// TwinCAT 3 PLC project PLC_Pro
// ProgramVersion: 3.1.4020.4
// libraries:
//   Tc2_MC2, * (Beckhoff Automation GmbH)
//   Tc2_Standard, * (Beckhoff Automation GmbH)
//   Tc2_System, * (Beckhoff Automation GmbH)
//   Tc3_Module, * (Beckhoff Automation GmbH)
//   VisuDialogs, * (System)
// project tree:
//   / GlobalTextList.TcGTLO, PlcTask.TcTTO, 视图管理器.TcVMO (not stored)
//   POUs/ MAIN.TcPOU
//   VISUs/ HMI.TcVIS
// real-time tasks:
//   TASK Task 1: cycle T#10ms, priority 1, ADS port 350
//   TASK PlcTask: cycle T#10ms, priority 20, ADS port 351
// motion (NC):
//   TASK NC-Task 1 SAF: cycle T#2ms, priority 4, ADS port 501
//   TASK NC-Task 1 SVB: cycle T#10ms, priority 8, ADS port 511
//   AXIS Axis 1 (id 1)
//     Velo: SlowManual=0.2, FastManual=1
//     OtherSettings: AllowMotionCmdToSlave=true, PulseDistancePos=0.5, PulseDistanceNeg=0.5
//     encoder EncType=19
//       EncPara: ScaleFactorNumerator=1, ScaleFactorDenominator=10000, Inverse=true, MaxCount=#xffffffff
//     drive DrvType=16
//       DrvPara: Inverse=true, MaxCount=#xffffffff
//         TimeComp: TaskDelayCycles=1
//     controller CtrType=1
//       CtrPara: PriorControlFactor=1
//         PosDiffControl: Enable=false
//         Observer: BandWidth=20
//   AXIS Axis 2 (id 2)
//     OtherSettings: AllowMotionCmdToSlave=true
//     encoder EncType=19
//       EncPara: ScaleFactorNumerator=5, ScaleFactorDenominator=10000, MaxCount=#xffffffff
//     drive DrvType=16
//       DrvPara: MaxCount=#xffffffff
//         TimeComp: TaskDelayCycles=1
//     controller CtrType=1
//       CtrPara: PriorControlFactor=1
//         PosDiffControl: Enable=false
//         Observer: BandWidth=20
//   AXIS Axis 3 (id 3)
//     OtherSettings: AllowMotionCmdToSlave=true
//     encoder EncType=19
//       EncPara: ScaleFactorNumerator=5, ScaleFactorDenominator=10000, Inverse=true, MaxCount=#xffffffff
//     drive DrvType=16
//       DrvPara: Inverse=true, MaxCount=#xffffffff
//         TimeComp: TaskDelayCycles=1
//     controller CtrType=1
//       CtrPara: PriorControlFactor=1
//         PosDiffControl: Enable=false
//         Observer: BandWidth=20
//   AXIS Axis 4 (id 4)
//     OtherSettings: AllowMotionCmdToSlave=true
//     encoder EncType=19
//       EncPara: ScaleFactorNumerator=360, ScaleFactorDenominator=10000, MaxCount=#xffffffff
//     drive DrvType=16
//       DrvPara: MaxCount=#xffffffff
//         TimeComp: TaskDelayCycles=1
//     controller CtrType=1
//       CtrPara: PriorControlFactor=1
//         Observer: BandWidth=20
//   AXIS Axis 5 (id 5)
//     OtherSettings: AllowMotionCmdToSlave=true
//     encoder EncType=19
//       EncPara: ScaleFactorNumerator=360, ScaleFactorDenominator=10000, MaxCount=#xffffffff
//     drive DrvType=16
//       DrvPara: MaxCount=#xffffffff
//         TimeComp: TaskDelayCycles=1
//     controller CtrType=1
//       CtrPara: PriorControlFactor=1
//         PosDiffControl: Enable=false
//         Observer: BandWidth=20
// I/O:
//   DEVICE Device 2 (EtherCAT), AmsNetId 169.254.52.53.3.1
//     Drive 1 (Elmo Drive) [Gold EtherCAT GCON Drive Rev:0x00010400]
//     Drive 2 (EP3E-EC) [EP3E-EC]
//     Drive 3 (EP3E-EC) [EP3E-EC]
//     Drive 4 (EP3E-EC) [EP3E-EC]
//     Drive 5 (EP3E-EC) [EP3E-EC]
// variable links:
//   NC-Task 1 SAF/Axes/Axis 1 <-> Device 2 (EtherCAT)/Drive 1 (Elmo Drive)
//     Drive/Inputs/In/nDcOutputTime <-> InfoData/DcOutputShift
//     Drive/Inputs/In/nState1 <-> Inputs/Status word
//     Drive/Inputs/In/nState2 <-> Inputs/Status word @bit 8
//     Drive/Inputs/In/nState4 @bit 1 <-> WcState/InputToggle
//     Drive/Inputs/In/nState4 <-> WcState/WcState
//     Drive/Outputs/Out/nCtrl1 <-> Outputs/Control word
//     Drive/Outputs/Out/nCtrl2 <-> Outputs/Control word @bit 8
//     Drive/Outputs/Out/nDataOut1 <-> Outputs/Target Position
//     Enc/Inputs/In/nDataIn1 <-> Inputs/Position actual value
//     Enc/Inputs/In/nDcInputTime <-> InfoData/DcInputShift
//     Enc/Inputs/In/nState4 @bit 1 <-> WcState/InputToggle
//     Enc/Inputs/In/nState4 <-> WcState/WcState
//   NC-Task 1 SAF/Axes/Axis 2 <-> Device 2 (EtherCAT)/Drive 2 (EP3E-EC)
//     Drive/Inputs/In/nDcOutputTime <-> InfoData/DcOutputShift
//     Drive/Inputs/In/nState1 <-> 2nd Transmit PDO mapping/Statusword
//     Drive/Inputs/In/nState2 <-> 2nd Transmit PDO mapping/Statusword @bit 8
//     Drive/Inputs/In/nState4 @bit 1 <-> WcState/InputToggle
//     Drive/Inputs/In/nState4 <-> WcState/WcState
//     Drive/Outputs/Out/nCtrl1 <-> 2nd Receive PDO mapping/Controlword
//     Drive/Outputs/Out/nCtrl2 <-> 2nd Receive PDO mapping/Controlword @bit 8
//     Drive/Outputs/Out/nDataOut1 <-> 2nd Receive PDO mapping/Target Position
//     Enc/Inputs/In/nDataIn1 <-> 2nd Transmit PDO mapping/Position Actual Value
//     Enc/Inputs/In/nDcInputTime <-> InfoData/DcInputShift
//     Enc/Inputs/In/nState4 @bit 1 <-> WcState/InputToggle
//     Enc/Inputs/In/nState4 <-> WcState/WcState
//   NC-Task 1 SAF/Axes/Axis 3 <-> Device 2 (EtherCAT)/Drive 3 (EP3E-EC)
//     Drive/Inputs/In/nDcOutputTime <-> InfoData/DcOutputShift
//     Drive/Inputs/In/nState1 <-> 2nd Transmit PDO mapping/Statusword
//     Drive/Inputs/In/nState2 <-> 2nd Transmit PDO mapping/Statusword @bit 8
//     Drive/Inputs/In/nState4 @bit 1 <-> WcState/InputToggle
//     Drive/Inputs/In/nState4 <-> WcState/WcState
//     Drive/Outputs/Out/nCtrl1 <-> 2nd Receive PDO mapping/Controlword
//     Drive/Outputs/Out/nCtrl2 <-> 2nd Receive PDO mapping/Controlword @bit 8
//     Drive/Outputs/Out/nDataOut1 <-> 2nd Receive PDO mapping/Target Position
//     Enc/Inputs/In/nDataIn1 <-> 2nd Transmit PDO mapping/Position Actual Value
//     Enc/Inputs/In/nDcInputTime <-> InfoData/DcInputShift
//     Enc/Inputs/In/nState4 @bit 1 <-> WcState/InputToggle
//     Enc/Inputs/In/nState4 <-> WcState/WcState
//   NC-Task 1 SAF/Axes/Axis 4 <-> Device 2 (EtherCAT)/Drive 4 (EP3E-EC)
//     Drive/Inputs/In/nDcOutputTime <-> InfoData/DcOutputShift
//     Drive/Inputs/In/nState1 <-> 2nd Transmit PDO mapping/Statusword
//     Drive/Inputs/In/nState2 <-> 2nd Transmit PDO mapping/Statusword @bit 8
//     Drive/Inputs/In/nState4 @bit 1 <-> WcState/InputToggle
//     Drive/Inputs/In/nState4 <-> WcState/WcState
//     Drive/Outputs/Out/nCtrl1 <-> 2nd Receive PDO mapping/Controlword
//     Drive/Outputs/Out/nCtrl2 <-> 2nd Receive PDO mapping/Controlword @bit 8
//     Drive/Outputs/Out/nDataOut1 <-> 2nd Receive PDO mapping/Target Position
//     Enc/Inputs/In/nDataIn1 <-> 2nd Transmit PDO mapping/Position Actual Value
//     Enc/Inputs/In/nDcInputTime <-> InfoData/DcInputShift
//     Enc/Inputs/In/nState4 @bit 1 <-> WcState/InputToggle
//     Enc/Inputs/In/nState4 <-> WcState/WcState
//   NC-Task 1 SAF/Axes/Axis 5 <-> Device 2 (EtherCAT)/Drive 5 (EP3E-EC)
//     Drive/Inputs/In/nDcOutputTime <-> InfoData/DcOutputShift
//     Drive/Inputs/In/nState1 <-> 2nd Transmit PDO mapping/Statusword
//     Drive/Inputs/In/nState2 <-> 2nd Transmit PDO mapping/Statusword @bit 8
//     Drive/Inputs/In/nState4 @bit 1 <-> WcState/InputToggle
//     Drive/Inputs/In/nState4 <-> WcState/WcState
//     Drive/Outputs/Out/nCtrl1 <-> 2nd Receive PDO mapping/Controlword
//     Drive/Outputs/Out/nCtrl2 <-> 2nd Receive PDO mapping/Controlword @bit 8
//     Drive/Outputs/Out/nDataOut1 <-> 2nd Receive PDO mapping/Target Position
//     Enc/Inputs/In/nDataIn1 <-> 2nd Transmit PDO mapping/Position Actual Value
//     Enc/Inputs/In/nDcInputTime <-> InfoData/DcInputShift
//     Enc/Inputs/In/nState4 @bit 1 <-> WcState/InputToggle
//     Enc/Inputs/In/nState4 <-> WcState/WcState
//   PLC_Pro/PLC_Pro Instance <-> NC-Task 1 SAF/Axes/Axis 1
//     PlcTask Inputs/MAIN.motor_Line.NcToPlc <-> Outputs/ToPlc
//     PlcTask Outputs/MAIN.motor_Line.PlcToNc <-> Inputs/FromPlc
//   PLC_Pro/PLC_Pro Instance <-> NC-Task 1 SAF/Axes/Axis 2
//     PlcTask Inputs/MAIN.motor_X.NcToPlc <-> Outputs/ToPlc
//     PlcTask Outputs/MAIN.motor_X.PlcToNc <-> Inputs/FromPlc
//   PLC_Pro/PLC_Pro Instance <-> NC-Task 1 SAF/Axes/Axis 3
//     PlcTask Inputs/MAIN.motor_Y.NcToPlc <-> Outputs/ToPlc
//     PlcTask Outputs/MAIN.motor_Y.PlcToNc <-> Inputs/FromPlc
//   PLC_Pro/PLC_Pro Instance <-> NC-Task 1 SAF/Axes/Axis 4
//     PlcTask Inputs/MAIN.motor_Angle.NcToPlc <-> Outputs/ToPlc
//     PlcTask Outputs/MAIN.motor_Angle.PlcToNc <-> Inputs/FromPlc
//   PLC_Pro/PLC_Pro Instance <-> NC-Task 1 SAF/Axes/Axis 5
//     PlcTask Inputs/MAIN.motor_Master.NcToPlc <-> Outputs/ToPlc
//     PlcTask Outputs/MAIN.motor_Master.PlcToNc <-> Inputs/FromPlc
//   TcAsyncBufferReadingDrv/ReadingModule <-> TcAsyncBufferReadingDrv/WriteDetect
//     Inputs/bExecute <-> Outputs/bExecuteOut
//     Inputs/nOffset <-> Outputs/nOffset
//   TcAsyncBufferReadingDrv/WriteDetect <-> TcAsyncBufferWritingDrv/WritingModule
//     Inputs/bBusy <-> Outputs/bBusy
//     Inputs/bError <-> Outputs/bError
//     Inputs/nBytesWritten <-> Outputs/nBytesWritten

CONFIGURATION PLC_Pro
    RESOURCE PLC ON TwinCAT3
        TASK PlcTask(INTERVAL := T#10ms, PRIORITY := 20);
        PROGRAM MAIN WITH PlcTask : MAIN;
    END_RESOURCE
END_CONFIGURATION

// ---- POUs/MAIN.TcPOU
PROGRAM MAIN
VAR
	power_On_motor_All                   :BOOL :=FALSE;   (*************)
	power_On_motor_Line                  :BOOL :=FALSE; 
	power_On_motor_X                     :BOOL :=FALSE; 
    power_On_motor_Y                     :BOOL :=FALSE; 
    power_On_motor_Angle                 :BOOL :=FALSE; 
    power_On_motor_Master                :BOOL :=FALSE; 
	
	
	move_do_Line                         :BOOL :=FALSE;   (*************)
	move_do_X                            :BOOL :=FALSE;
	move_do_Y                            :BOOL :=FALSE;
    move_do_Angle                        :BOOL :=FALSE;
    move_do_Master                       :BOOL :=FALSE;
	
	set_do_Line                         :BOOL :=FALSE;    (*************)
	set_do_X                            :BOOL :=FALSE;
	set_do_Y                            :BOOL :=FALSE;
    set_do_Angle                        :BOOL :=FALSE;
    set_do_Master                       :BOOL :=FALSE;
	
	stop_do_Line                         :BOOL :=FALSE;
	stop_do_X                            :BOOL :=FALSE;
	stop_do_Y                            :BOOL :=FALSE;
    stop_do_Angle                        :BOOL :=FALSE;
    stop_do_Master                       :BOOL :=FALSE;
	
	reset_do_Line                         :BOOL :=FALSE;
	reset_do_X                            :BOOL :=FALSE;
	reset_do_Y                            :BOOL :=FALSE;
    reset_do_Angle                        :BOOL :=FALSE;
    reset_do_Master                       :BOOL :=FALSE;
	
	move_r_INC_motor_Line                 : REAL       :=0;   (****定义运动增量****)
	move_r_INC_motor_X                    : REAL       :=0;   (****关联到HMI界面****)
	move_r_INC_motor_Y                    : REAL       :=0;
	move_r_INC_motor_Angle                : REAL       :=0;
	move_r_INC_motor_Master               : REAL       :=0;
	
	(***定义轴变量***)
	motor_Line , motor_X , motor_Y , motor_Angle , motor_Master    :axis_ref;  (***定义轴变量***)
	(*****定义电源控制变量*****)
	mc_power_Line , mc_power_X , mc_power_Y , mc_power_Angle , mc_power_Master    :mc_power;   
	(****定义轴增量运动功能块*****)
	move_r_Line,  move_r_X,  move_r_Y,  move_r_Angle, move_r_Master   :mc_MoveRelative; 
	(******定义轴当前位置*****)
	position_Line, position_X, position_Y, 	position_Angle, position_Master  :mc_setposition; 
	(******定义轴停止*****) 
    stop_Line, stop_X, stop_Y, 	stop_Angle, stop_Master  :mc_stop;  
	(******定义轴复位*****)
    reset_Line, reset_X, reset_Y, reset_Angle, reset_Master  :mc_reset;  
	
END_VAR

(***********定义直线电机电源************)
mc_power_Line(
	Axis:= motor_Line, 
	Enable:= power_On_motor_All AND power_On_motor_Line, 
	Enable_Positive:= TRUE , 
	Enable_Negative:= TRUE, 
//	Override:= , 
//	BufferMode:= , 
//	Options:= , 
//	Status=> , 
//	Busy=> , 
//	Active=> , 
//	Error=> , 
//	ErrorID=> 
);
(***********定义X轴电机电源************)
	mc_power_X(
	Axis:=motor_X , 
	Enable:=power_On_motor_All AND  power_On_motor_X, 
	Enable_Positive:= TRUE, 
	Enable_Negative:= TRUE, 
	Override:= , 
	BufferMode:= , 
	Options:= , 
	Status=> , 
	Busy=> , 
	Active=> , 
	Error=> , 
	ErrorID=> );

(***********定义Y轴电机电源************)	
	mc_power_Y(
	Axis:= motor_Y, 
	Enable:= power_On_motor_All AND power_On_motor_Y, 
	Enable_Positive:= TRUE , 
	Enable_Negative:= TRUE , 
	Override:= , 
	BufferMode:= , 
	Options:= , 
	Status=> , 
	Busy=> , 
	Active=> , 
	Error=> , 
	ErrorID=> );
	
(***********定义摆角电机电源************)	
	mc_power_Angle(
	Axis:= motor_Angle, 
	Enable:=power_On_motor_All AND  power_On_motor_Angle, 
	Enable_Positive:= TRUE, 
	Enable_Negative:= TRUE, 
	Override:= , 
	BufferMode:= , 
	Options:= , 
	Status=> , 
	Busy=> , 
	Active=> , 
	Error=> , 
	ErrorID=> );
	
(***********定义主轴电机电源************)
	mc_power_Master(
	Axis:= motor_Master, 
	Enable:= power_On_motor_All AND   power_On_motor_Master, 
	Enable_Positive:= TRUE, 
	Enable_Negative:= TRUE, 
	Override:= , 
	BufferMode:= , 
	Options:= , 
	Status=> , 
	Busy=> , 
	Active=> , 
	Error=> , 
	ErrorID=> );
	
(***********定义直线电机运动************)
	move_r_Line(
	Axis:= motor_X, 
	Execute:= move_do_X, 
	Distance:= 1, 
	Velocity:=1 , 
	Acceleration:= , 
	Deceleration:= , 
	Jerk:= , 
	BufferMode:= , 
	Options:= , 
	Done=> , 
	Busy=> , 
	Active=> , 
	CommandAborted=> , 
	Error=> , 
	ErrorID=> );
	
(***********定义X轴电机运动************)
	move_r_X(
	Axis:= motor_X, 
	Execute:= move_do_X, 
	Distance:= aa, 
	Velocity:= 1, 
	Acceleration:= , 
	Deceleration:= , 
	Jerk:= , 
	BufferMode:= , 
	Options:= , 
	Done=> , 
	Busy=> , 
	Active=> , 
	CommandAborted=> , 
	Error=> , 
	ErrorID=> );
	
(***********定义Y轴电机运动************)
	move_r_Y(
	Axis:= motor_Y, 
	Execute:= move_do_Y, 
	Distance:= 1, 
	Velocity:= 1, 
	Acceleration:= , 
	Deceleration:= , 
	Jerk:= , 
	BufferMode:= , 
	Options:= , 
	Done=> , 
	Busy=> , 
	Active=> , 
	CommandAborted=> , 
	Error=> , 
	ErrorID=> );
	
(***********定义摆角电机运动************)
	move_r_Angle(
	Axis:= motor_Angle, 
	Execute:= move_do_Angle, 
	Distance:=1 , 
	Velocity:= 1, 
	Acceleration:= , 
	Deceleration:= , 
	Jerk:= , 
	BufferMode:= , 
	Options:= , 
	Done=> , 
	Busy=> , 
	Active=> , 
	CommandAborted=> , 
	Error=> , 
	ErrorID=> );
	
(***********定义主轴电机运动************)
	move_r_Master(
	Axis:= motor_Master, 
	Execute:= move_do_Master, 
	Distance:=1 , 
	Velocity:= 1, 
	Acceleration:= , 
	Deceleration:= , 
	Jerk:= , 
	BufferMode:= , 
	Options:= , 
	Done=> , 
	Busy=> , 
	Active=> , 
	CommandAborted=> , 
	Error=> , 
	ErrorID=> );

(***********定义直线电机当前位置************)	
	position_Line(
	Axis:=motor_Line , 
	Execute:= set_do_Line, 
	Position:= 0, 
	Mode:= , 
	Options:= , 
	Done=> , 
	Busy=> , 
	Error=> , 
	ErrorID=> );

(***********定义X轴电机当前位置************)	
	position_X(
	Axis:= motor_X , 
	Execute:= set_do_X , 
	Position:= 0, 
	Mode:= , 
	Options:= , 
	Done=> , 
	Busy=> , 
	Error=> , 
	ErrorID=> );
	
(***********定义y轴电机当前位置************)	
	position_Y(
	Axis:= motor_Y , 
	Execute:= set_do_Y , 
	Position:= 0, 
	Mode:= , 
	Options:= , 
	Done=> , 
	Busy=> , 
	Error=> , 
	ErrorID=> );
	
(***********定义摆角电机当前位置************)	
	position_Angle(
	Axis:= motor_Angle , 
	Execute:= set_do_Angle , 
	Position:= 0, 
	Mode:= , 
	Options:= , 
	Done=> , 
	Busy=> , 
	Error=> , 
	ErrorID=> );
	
(***********定义主轴电机当前位置************)	
	position_Master(
	Axis:= motor_Master , 
	Execute:= set_do_Master , 
	Position:= 0, 
	Mode:= , 
	Options:= , 
	Done=> , 
	Busy=> , 
	Error=> , 
	ErrorID=> );

(***********定义直线电机停止************)	
	stop_Line(
	Axis:= motor_Line , 
	Execute:= stop_do_Line, 
	Deceleration:= , 
	Jerk:= , 
	Options:= , 
	Done=> , 
	Busy=> , 
	Active=> , 
	CommandAborted=> , 
	Error=> , 
	ErrorID=> );
	
	(***********定义X轴电机停止************)	
	stop_X(
	Axis:= motor_X , 
	Execute:= stop_do_X, 
	Deceleration:= , 
	Jerk:= , 
	Options:= , 
	Done=> , 
	Busy=> , 
	Active=> , 
	CommandAborted=> , 
	Error=> , 
	ErrorID=> );

(***********定义Y轴电机停止************)	
	stop_Y(
	Axis:= motor_Y , 
	Execute:= stop_do_Y, 
	Deceleration:= , 
	Jerk:= , 
	Options:= , 
	Done=> , 
	Busy=> , 
	Active=> , 
	CommandAborted=> , 
	Error=> , 
	ErrorID=> );
	
(***********定义摆角电机停止************)	
	stop_Angle(
	Axis:= motor_Angle , 
	Execute:= stop_do_Angle, 
	Deceleration:= , 
	Jerk:= , 
	Options:= , 
	Done=> , 
	Busy=> , 
	Active=> , 
	CommandAborted=> , 
	Error=> , 
	ErrorID=> );
	
(***********定义主轴电机停止************)	
	stop_Master(
	Axis:= motor_Master , 
	Execute:= stop_do_Master, 
	Deceleration:= , 
	Jerk:= , 
	Options:= , 
	Done=> , 
	Busy=> , 
	Active=> , 
	CommandAborted=> , 
	Error=> , 
	ErrorID=> );

(***********定义直线电机复位************)	
	reset_Line(
	Axis:= motor_Line, 
	Execute:= reset_do_Line, 
	Done=> , 
	Busy=> , 
	Error=> , 
	ErrorID=> );
	
(***********定义X轴电机复位************)	
	reset_X(
	Axis:= motor_X, 
	Execute:= reset_do_X, 
	Done=> , 
	Busy=> , 
	Error=> , 
	ErrorID=> );
	
(***********定义Y轴电机复位************)	
	reset_Y(
	Axis:= motor_Y, 
	Execute:= reset_do_Y, 
	Done=> , 
	Busy=> , 
	Error=> , 
	ErrorID=> );
	
(***********定义摆角电机复位************)	
	reset_Angle(
	Axis:= motor_Angle, 
	Execute:= reset_do_Angle, 
	Done=> , 
	Busy=> , 
	Error=> , 
	ErrorID=> );
	
(***********定义主轴电机复位************)	
	reset_Master(
	Axis:= motor_Master, 
	Execute:= reset_do_Master, 
	Done=> , 
	Busy=> , 
	Error=> , 
	ErrorID=> );

END_PROGRAM

// ---- GlobalTextList.TcGTLO
TEXTLIST GlobalTextList
  41 = '%.2f'
  43 = '%.6f'
  47 = 'INC_Angle%.6f'
  44 = 'INC_Line%.6f'
  45 = 'INC_X%.6f'
  46 = 'INC_Y%.6f'
  39 = 'motorAngle:%.2f'
  36 = 'motorLine:%.2f'
  42 = 'motorLine_INC%.6f'
  40 = 'motorMaster:%.2f'
  37 = 'motorX:%.2f'
  38 = 'motorY:%.2f'
  4 = 'motor_Angle'
  7 = 'motor_Angle:%.2f'
  0 = 'motor_Line:%.2f'
  5 = 'motor_Master:'
  6 = 'motor_Master:%.2f'
  1 = 'motor_X:%.2f'
  2 = 'motor_Y'
  3 = 'motor_Y:%.2f'
  18 = 'MoveReAngle'
  15 = 'MoveReLine'
  19 = 'MoveReMaster'
  16 = 'MoveReX'
  17 = 'MoveReY'
  23 = 'PositionAngle'
  20 = 'PositionLine'
  24 = 'PositionMaster'
  21 = 'PositionX'
  22 = 'PositionY'
  9 = 'PowerOnAll'
  13 = 'PowerOnAngle'
  10 = 'PowerOnLine'
  14 = 'PowerOnMaster'
  11 = 'PowerOnX'
  12 = 'PowerOnY'
  8 = 'power_On_motor_All'
  34 = 'ResetAngle'
  31 = 'ResetLine'
  35 = 'ResetMaster'
  32 = 'ResetX'
  33 = 'ResetY'
  29 = 'StopAngle'
  26 = 'StopLine'
  30 = 'StopMaster'
  28 = 'StopX'
  27 = 'StopY'
  25 = 'stop_Line'
END_TEXTLIST

// ---- VISUs/HMI.TcVIS
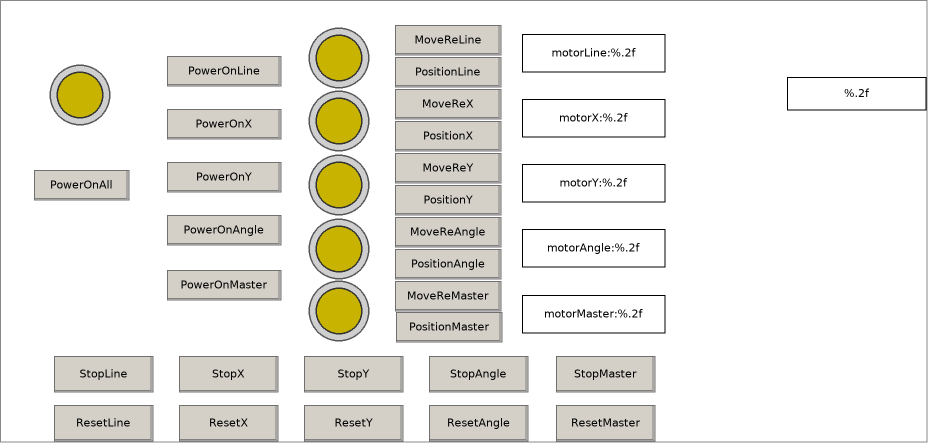
VISUALIZATION HMI  // 928x443
    Group (34,23 631x418)
        Rectangle (488,11 143x38), "motorLine:%.2f", text variable: MAIN.motor_Line.NcToPlc.ActPos
        Rectangle (488,272 143x38), "motorMaster:%.2f", text variable: MAIN.motor_Master.NcToPlc.ActPos
        Rectangle (488,76 143x38), "motorX:%.2f", text variable: MAIN.motor_X.NcToPlc.ActPos
        Rectangle (488,141 143x38), "motorY:%.2f", text variable: MAIN.motor_Y.NcToPlc.ActPos
        Rectangle (488,206 143x38), "motorAngle:%.2f", text variable: MAIN.motor_Angle.NcToPlc.ActPos
        Lamp1 (270,0 70x70), variable: MAIN.motor_Line.NcToPlc.StateDWord.20, style: Lamp-Lamp1-Yellow
        Lamp1 (270,63 70x70), variable: MAIN.motor_X.NcToPlc.StateDWord.20, style: Lamp-Lamp1-Yellow
        Lamp1 (270,127 70x70), variable: MAIN.motor_Y.NcToPlc.StateDWord.20, style: Lamp-Lamp1-Yellow
        Lamp1 (270,191 70x70), variable: MAIN.motor_Angle.NcToPlc.StateDWord.20, style: Lamp-Lamp1-Yellow
        Lamp1 (270,253 70x70), variable: MAIN.motor_Master.NcToPlc.StateDWord.20, style: Lamp-Lamp1-Yellow
        Lamp1 (11,37 70x70), variable: MAIN.power_On_motor_All, style: Lamp-Lamp1-Yellow
        Button (0,147 95x30), "PowerOnAll", text variable: MAIN.power_On_motor_All
            toggle MAIN.power_On_motor_All
        Button (133,33 114x30), "PowerOnLine"
            toggle MAIN.power_On_motor_Line
        Button (133,192 114x30), "PowerOnAngle"
            toggle MAIN.power_On_motor_Angle
        Button (133,139 114x30), "PowerOnY"
            toggle MAIN.power_On_motor_Y
        Button (133,86 114x30), "PowerOnX"
            toggle MAIN.power_On_motor_X
        Button (133,247 114x30), "PowerOnMaster"
            toggle MAIN.power_On_motor_Master
        Button (361,2 106x30), "MoveReLine"
            tap MAIN.move_do_Line
        Button (361,34 106x30), "PositionLine"
            tap MAIN.set_do_Line
        Button (361,66 106x30), "MoveReX"
            tap MAIN.move_do_X
        Button (361,98 106x30), "PositionX"
            tap MAIN.set_do_X
        Button (361,194 106x30), "MoveReAngle"
            tap MAIN.move_do_Angle
        Button (361,162 106x30), "PositionY"
            tap MAIN.set_do_Y
        Button (361,130 106x30), "MoveReY"
            tap MAIN.move_do_Y
        Button (361,226 106x30), "PositionAngle"
            tap MAIN.set_do_Angle
        Button (361,258 106x30), "MoveReMaster"
            tap MAIN.move_do_Master
        Button (362,289 106x30), "PositionMaster"
            tap MAIN.set_do_Master
        Button (20,333 99x36), "StopLine"
            tap MAIN.stop_do_Line
        Button (145,333 99x36), "StopX"
            tap MAIN.stop_do_X
        Button (270,333 99x36), "StopY"
            tap MAIN.stop_do_Y
        Button (395,333 99x36), "StopAngle"
            tap MAIN.stop_do_Angle
        Button (522,333 99x36), "StopMaster"
            tap MAIN .stop_do_Master
        Button (20,382 99x36), "ResetLine"
            tap MAIN.reset_do_Line
        Button (145,382 99x36), "ResetX"
            tap MAIN.reset_do_X
        Button (270,382 99x36), "ResetY"
            tap MAIN.reset_do_Y
        Button (395,382 99x36), "ResetAngle"
            tap MAIN.reset_do_Angle
        Button (522,382 99x36), "ResetMaster"
            tap MAIN.reset_do_Master
    Rectangle (787,77 139x33), "%.2f", text variable: MAIN.aa
        OnMouseDown: write the text variable via Default
END_VISUALIZATION
